(* Schneider Machine Expert - Basic project Motor_Full_TM221CE16T, file version 3.0.0.0 *)
(* ProjectInformations: Name=New project *)

HARDWARE
  Cpu 0: TM221CE16T
  EthernetConfiguration: NetworkName=M221, IpAllocationMode=FixedAddress, IpAddress=0.0.0.0, SubnetMask=0.0.0.0
  SerialLineConfiguration: Baud=Baud19200, Parity=ParityEven, DataBits=DataBits8, StopBits=StopBits1, PhysicalMedium=PhysicalMediumRs485, TransmissionMode=TransmissionModeModbusRtu, SlaveId=1, Addressing=SlaveAddressing
  MastTask: UsePeriodScanMode=false, PeriodScan=100
  FastTask: Period=255
  CpuBehavior: StartingMode=StartAsPreviousState, AutoSaveRamOnEeprom=true, WatchdogPeriod=250

SYMBOLS  (address, symbol, comment, settings)
  %M0       SYSTEM_READY
  %S0       SB_COLDSTART  "Indicates or executes a cold start (data initialized to default values)"
  %S1       SB_WARMSTART  "Indicates there was a warm start with data backup"
  %TM0        [Preset=3, Base=OneSecond]
  %I0.0     EMERGENCY_PB

POU New POU
  (* SectionNumber=0 *)

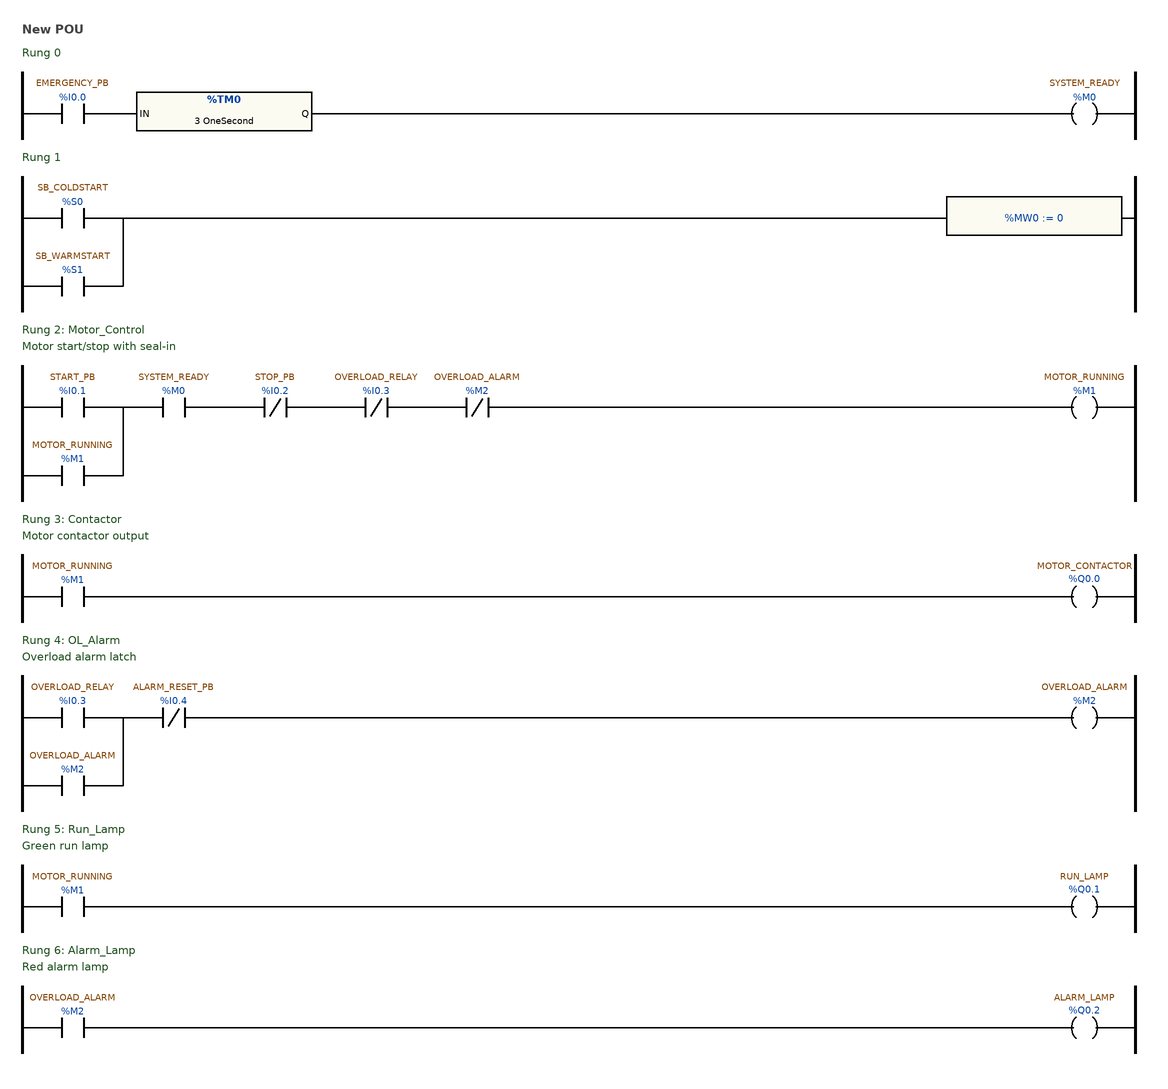

// Rung 0
  BLK %TM0
  LD %I0.0                (* EMERGENCY_PB *)
  IN
  OUT_BLK
  LD Q
  ST %M0                  (* SYSTEM_READY *)
  END_BLK
  // as ST:
  //   %TM0(IN := EMERGENCY_PB);
  //   SYSTEM_READY := %TM0.Q;

// Rung 1
  LD %S0                  (* SB_COLDSTART *)
  OR %S1                  (* SB_WARMSTART *)
  [ %MW0 := 0 ]
  // as ST:
  //   IF SB_COLDSTART OR SB_WARMSTART THEN %MW0 := 0; END_IF;

// Rung 2: Motor_Control
// Motor start/stop with seal-in
  LD %I0.1
  OR %M1
  AND %M0                 (* SYSTEM_READY *)
  ANDN %I0.2
  ANDN %I0.3
  ANDN %M2
  ST %M1
  // %I0.1: Start Button
  // %M0: System Ready
  // %I0.2: Stop NC
  // %I0.3: Overload OK
  // %M2: No Alarm
  // %M1: Motor Run
  // %M1: Seal-in
  // as ST:
  //   %M1 := (%I0.1 OR %M1) AND SYSTEM_READY AND NOT %I0.2 AND NOT %I0.3 AND NOT %M2;

// Rung 3: Contactor
// Motor contactor output
  LD %M1
  ST %Q0.0
  // %M1: Motor Running
  // %Q0.0: Contactor
  // as ST:
  //   %Q0.0 := %M1;

// Rung 4: OL_Alarm
// Overload alarm latch
  LD %I0.3
  OR %M2
  ANDN %I0.4
  ST %M2
  // %I0.3: Overload Trip
  // %I0.4: Reset
  // %M2: Alarm
  // %M2: Latch
  // as ST:
  //   %M2 := (%I0.3 OR %M2) AND NOT %I0.4;

// Rung 5: Run_Lamp
// Green run lamp
  LD %M1
  ST %Q0.1
  // %M1: Running
  // %Q0.1: Run Lamp
  // as ST:
  //   %Q0.1 := %M1;

// Rung 6: Alarm_Lamp
// Red alarm lamp
  LD %M2
  ST %Q0.2
  // %M2: Alarm
  // %Q0.2: Alarm Lamp
  // as ST:
  //   %Q0.2 := %M2;

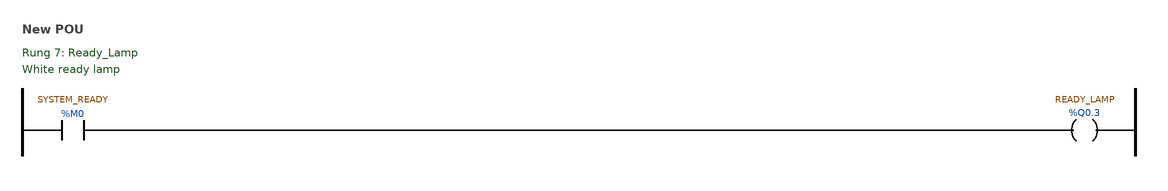

// Rung 7: Ready_Lamp
// White ready lamp
  LD %M0                  (* SYSTEM_READY *)
  ST %Q0.3
  // %M0: Ready
  // %Q0.3: Ready Lamp
  // as ST:
  //   %Q0.3 := SYSTEM_READY;
